// TIA Portal V17 export
// export: Created 2024-08-09T12:53:23.360791Z, ExportSetting WithDefaults, DisplayName Totally Integrated Automation Portal, DisplayVersion V17 Update 7, DisplayName TIA Portal Openness, DisplayVersion V17 Update 7, DisplayName TIA Portal Version Control Interface, DisplayVersion V17, DisplayName STEP 7 Professional, DisplayVersion V17 Update 7, DisplayName STEP 7 Safety, DisplayVersion V17 Update 6, DisplayName WinCC Professional, DisplayVersion V17 Update 7
TYPE "S_Compo_char"
// stored: IsFailsafeCompliant false
   STRUCT
      _PtcelOrigPrec { ExternalAccessible := 'False'; ExternalVisible := 'False'; ExternalWritable := 'False'} : "S_Cellule";   // cellule precedente
      _NoLotOrig { ExternalAccessible := 'False'; ExternalVisible := 'False'; ExternalWritable := 'False'} : String["T_Num_Lot"];   // Numero de lot
      _CdMat { ExternalAccessible := 'False'; ExternalVisible := 'False'; ExternalWritable := 'False'} : String["T_CD_MAT"];   // code mp
      _LbMat { ExternalAccessible := 'False'; ExternalVisible := 'False'; ExternalWritable := 'False'} : String["T_LB_MAT"];   // libelle mp
      _CdMatOrg { ExternalAccessible := 'False'; ExternalVisible := 'False'; ExternalWritable := 'False'} : String["T_CD_MAT"];   // code mp Equivalente
      _LbMatOrg { ExternalAccessible := 'False'; ExternalVisible := 'False'; ExternalWritable := 'False'} : String["T_LB_MAT"];   // libelle mp Equivalente
      _CdProc { ExternalAccessible := 'False'; ExternalVisible := 'False'; ExternalWritable := 'False'} : String["T_PROC"];
      _Presentation { ExternalAccessible := 'False'; ExternalVisible := 'False'; ExternalWritable := 'False'} : String["T_PRESENT"];
      _PProc { ExternalAccessible := 'False'; ExternalVisible := 'False'; ExternalWritable := 'False'} : String["T_PROC"];
      _CdForm { ExternalAccessible := 'False'; ExternalVisible := 'False'; ExternalWritable := 'False'} : String["T_CD_FOR"];   // code formule
      _LibFor { ExternalAccessible := 'False'; ExternalVisible := 'False'; ExternalWritable := 'False'} : String["T_LB_FOR"];   // libelle formule
      _Version { ExternalAccessible := 'False'; ExternalVisible := 'False'; ExternalWritable := 'False'} : String["T_CD_VER"];   // code version
      _Repart { ExternalAccessible := 'False'; ExternalVisible := 'False'; ExternalWritable := 'False'} : String["T_CD_REP"];   // code repartition
      _EtatChar { ExternalAccessible := 'False'; ExternalVisible := 'False'; ExternalWritable := 'False'} : Char;   // Etat du fin de chargement ('O', 'N', 'C')
      _Pourcent { ExternalAccessible := 'False'; ExternalVisible := 'False'; ExternalWritable := 'False'} : Real;   // pourcentage a incorporer
      _PoidsRestant { ExternalAccessible := 'False'; ExternalVisible := 'False'; ExternalWritable := 'False'} : Real;   // poids restant a doser si multi pesees
      _QteBrut : Real;   // quantite brut
      _ConsQte : Real;   // poids a dosee pour la pesee
      _ConsArret : Real;   // Consigne d'arret
      _QteNet : Real;   // poids Net
      _QteDejaChargee : Real;   // poids deja chargee
      _QteMvt { ExternalAccessible := 'False'; ExternalVisible := 'False'; ExternalWritable := 'False'} : Real;   // poids deja mouvemente
      _TareCel { ExternalAccessible := 'False'; ExternalVisible := 'False'; ExternalWritable := 'False'} : Real;   // Tare composant cellule
      _Ecart : Real;   // Ecart dosage composant en kilos
      _Vitesse { ExternalAccessible := 'False'; ExternalVisible := 'False'; ExternalWritable := 'False'} : Real;   // Vitesse
      _NoPeseeTare { ExternalAccessible := 'False'; ExternalVisible := 'False'; ExternalWritable := 'False'} : USInt;   // numero de pesee Tare
      _NoPeseeBrut { ExternalAccessible := 'False'; ExternalVisible := 'False'; ExternalWritable := 'False'} : USInt;   // numero de pesee Brut
      _Case : USInt;
      _FgAbandon { ExternalAccessible := 'False'; ExternalVisible := 'False'; ExternalWritable := 'False'} : Bool;   // Abandon dosage composant
      _FgFincharg { ExternalAccessible := 'False'; ExternalVisible := 'False'; ExternalWritable := 'False'} : Bool;   // Dosage composant termine
      _FgSeq { ExternalAccessible := 'False'; ExternalVisible := 'False'; ExternalWritable := 'False'} : Bool;   // Flag sequence ouv/ferm vide cellule effectue
      _FgTareConnue { ExternalAccessible := 'False'; ExternalVisible := 'False'; ExternalWritable := 'False'} : Bool;   // Flag tare connue
      _FgCelluleVide { ExternalAccessible := 'False'; ExternalVisible := 'False'; ExternalWritable := 'False'} : Bool;   // flag cellule vide
      _FgaVider { ExternalAccessible := 'False'; ExternalVisible := 'False'; ExternalWritable := 'False'} : Bool;   // flag de demande de vide cellule
      _FgCb { ExternalAccessible := 'False'; ExternalVisible := 'False'; ExternalWritable := 'False'} : Bool;   // flag Code Barre
   END_STRUCT;
END_TYPE
